PROGRAM BH0GPL_LineBackground
VAR
END_VAR

MAIN.stLine_BH0GPL.fbLine(stLine:=MAIN.stLine_BH0GPL);
MAIN.stLine_BH0GPL.stStation_BH0GPL01.fbStation(
				stLine:=MAIN.stLine_BH0GPL,
				stStation:=MAIN.stLine_BH0GPL.stStation_BH0GPL01);

END_PROGRAM

(* stored: Version 1.1.0.1, ProductVersion 3.1.4024.15
   POU BH0GPL_LineBackground: Id {a680d076-a87f-416e-9aea-1c311db5fc5b}, SpecialFunc None *)
